Fanuc KAREL source: NC0074.KL

-- PROVISIONAL review KL for V1013-1; original PC SHA256 ca0fb687aabaedd0dc0f4309cd80b0df89c10e2b2e6b3c365b871e190c99cbc5
-- Incomplete behavior may be omitted. Consult companion uncertainty JSON. Do not deploy.
PROGRAM NC0074
%NOLOCKGROUP
-- UNRESOLVED_LOCAL_POOL 1 cells at code offset 3; source declarations unknown
-- DIRECT_LOCAL_WORD_ACCESS alone does not prove INTEGER, REAL, or BOOLEAN
BEGIN
  -- UNRESOLVED_PC offsets 0-8; opcodes 2B,2C,7B
  -- UNRESOLVED_PC offsets 13-20; opcodes 9D,23
  -- UNRESOLVED_PC offsets 25-42; opcodes 21,2E,59,79
  -- UNRESOLVED_PC offsets 47-64; opcodes 21,2E,59,79
  -- UNRESOLVED_PC offsets 69-86; opcodes 21,2E,59,79
  -- UNRESOLVED_PC offsets 91-105; opcodes 21,9D,52,23
  -- UNRESOLVED_PC offsets 110-115; opcodes 7A
  -- UNRESOLVED_PC offsets 120-125; opcodes 7A
  -- UNRESOLVED_PC offsets 130-135; opcodes 7A
  -- UNRESOLVED_PC offsets 140-144; opcodes 7F
  -- UNRESOLVED_PC offsets 149-153; opcodes 27,AA
  -- UNRESOLVED_PC offsets 158-162; opcodes 7F
END NC0074
